FUNCTION F_Scaling : REAL
VAR_INPUT

	nAnalogIn								:INT;
	fNumerator								:REAL;
	fDenominator							:REAL;
	
END_VAR
VAR
END_VAR
(* End *)

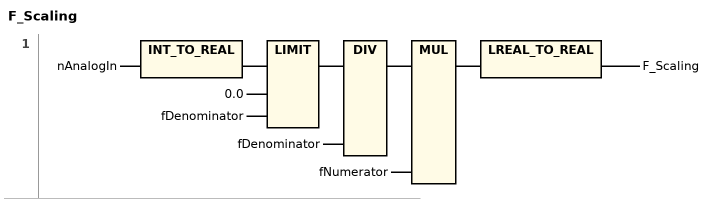
// NETWORK 1
F_Scaling := LREAL_TO_REAL((LIMIT(INT_TO_REAL(nAnalogIn), 0.0, fDenominator) / fDenominator) * fNumerator);

END_FUNCTION

(* stored: Version 1.1.0.1, ProductVersion 3.1.4018.5
   POU F_Scaling: Id {d72d2195-0754-4efc-8911-b16247d2b396}, SpecialFunc None *)
